// TIA Portal project "Automated Door with Delay" (V17)
// Automated Door with Delay
// The motion sensor detects when someone approaching the door, should wait for 10 sec and then open. If no one is detected for 5 sec, the door should close.

(* hardware
DEVICE "S7-1200 station_1"  S7-1200 Station
   slot 0: "Rack_0"  S7-1200 Rack  Rack  V1.0
   slot 1: "PLC_1"  CPU 1214C AC/DC/Rly  6ES7 214-1BG40-0XB0  V4.5
*)

// ===== PLC "PLC_1"  CPU 1214C AC/DC/Rly =====

VAR_GLOBAL   // PLC tag table "Default tag table"
   "Start_Button" AT %I0.0 : Bool;
   "Motion_Sensor" AT %I0.1 : Bool;
   "Door_Locked" AT %Q0.0 : Bool;
   "Tag_1" AT %M0.0 : Bool;
END_VAR

// folder: System blocks/Program resources

DATA_BLOCK "IEC_Timer_0_DB"   // DB1
{ S7_Optimized_Access := 'TRUE' }
AUTHOR : Simatic
FAMILY : IEC
NAME : IEC_TMR
VERSION : 1.0
// stored: InstanceOfName IEC_TIMER
"IEC_TIMER"
BEGIN
END_DATA_BLOCK

DATA_BLOCK "IEC_Timer_0_DB_1"   // DB2
{ S7_Optimized_Access := 'TRUE' }
AUTHOR : Simatic
FAMILY : IEC
NAME : IEC_TMR
VERSION : 1.0
// stored: InstanceOfName IEC_TIMER
"IEC_TIMER"
BEGIN
END_DATA_BLOCK

// folder: (top level)

ORGANIZATION_BLOCK "Main"   // OB1, LAD, ProgramCycle
TITLE = "Main Program Sweep (Cycle)"
{ S7_Optimized_Access := 'TRUE' }
VERSION : 0.1
   VAR_INPUT
      Initial_Call : Bool;   // Initial call of this OB
      Remanence : Bool;   // =True, if remanent data are available
   END_VAR
BEGIN

REGION Network 1
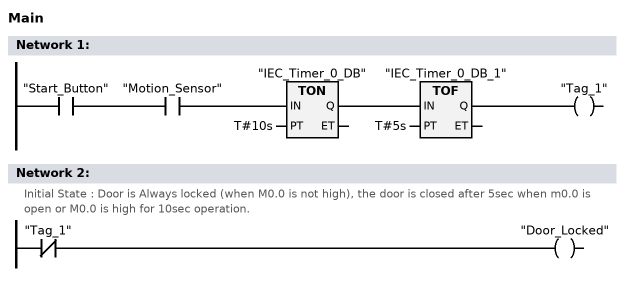
   "IEC_Timer_0_DB".TON(IN := "Start_Button" AND "Motion_Sensor", PT := T#10s);
   "IEC_Timer_0_DB_1".TOF(IN := "IEC_Timer_0_DB".Q, PT := T#5s);
   "Tag_1" := "IEC_Timer_0_DB_1".Q;
END_REGION

REGION Network 2
   // Initial State : Door is Always locked (when M0.0 is not high), the door is closed after 5sec when m0.0 is open or M0.0 is high for 10sec operation.
   RUNG wire#powerrail
      I_Contact( "Tag_1" )
      Coil( "Door_Locked" )
   END_RUNG
   // the same network as SCL:
   "Door_Locked" := NOT "Tag_1";
END_REGION
END_ORGANIZATION_BLOCK